FUNCTION_BLOCK MockSerializableArray IMPLEMENTS I_Serializable
VAR
	_name : STRING;
	_age : INT;
END_VAR

PROPERTY PUBLIC Age : INT
GET
Age := _age;
END_GET
SET
_age := Age;
END_SET
END_PROPERTY

METHOD FB_init : BOOL
VAR_INPUT
	bInitRetains : BOOL; // if TRUE, the retain variables are initialized (warm start / cold start)
	bInCopyCode : BOOL;  // if TRUE, the instance afterwards gets moved into the copy code (online change)
	Name : STRING;
	Age : INT;
END_VAR
_name := Name;
_age := Age;
END_METHOD

PROPERTY PUBLIC Name : STRING
GET
Name := _name;
END_GET
SET
_name := Name;
END_SET
END_PROPERTY

METHOD SerializeWith
VAR_INPUT
	Serializer : I_Serializer;
END_VAR
Serializer.StartArray().AddString(_name).AddInt(_age).EndArray();
END_METHOD

END_FUNCTION_BLOCK

(* stored: Version 1.1.0.1, ProductVersion 3.1.4024.12
   POU MockSerializableArray: Id {1699a081-b0e6-403b-be67-114f85fe3b83}, SpecialFunc None
   Folder Constructor: Id {349edc1d-7b42-4dbb-ae41-98cb7d508241}
   Property Age: Id {81fd92af-dcaa-4599-b7c2-dea7e9db55ad}
   Get Get: Id {7ddce9be-537e-46ae-81dc-3fdb86ad0e21}
   Set Set: Id {db6a5458-9903-450f-8a13-d9aef6ba7db4}
   Method FB_init: Id {aed1f564-7d32-48e9-a351-469346c2e14b}
   Property Name: Id {fa65ec32-6bdd-4566-888b-5cbf9f40c471}
   Get Get: Id {86233638-af6f-4d92-8526-17980efbf873}
   Set Set: Id {c41bc441-815c-4f50-a4c4-e70adf12c2a9}
   Method SerializeWith: Id {ee5c045e-7d52-43c1-bea9-d41685013b96} *)
